{attribute 'qualified_only'}
{attribute 'strict'}
{attribute 'to_string'}
TYPE E_TrackName :
(
	T1_1_ToRotate := 1,
	T1_2_ToBranch,
	T2_1_ToLink,
	T2_2_ToRotate,
	T2_3_ToEnd,
	T3_1_ToLink,
	T3_2_ToRotate,
	T3_3_ToEnd
);
END_TYPE

(* stored: Version 1.1.0.1
   DUT E_TrackName: Id {5eca3b88-723a-4757-8d39-6432a19566fd} *)
